(* IEC 61131-3 sources: com.logicals.lc3.webinar/RPMControl_Webinar/src_PRG_MQTT_Raspi2_ST, 4 files *)

(* ---- PRG_Raspi2_MQTTConnect.iecst ---- *)
/*
 * Raspi2
 * MQTTConnect Task
 */
PROGRAM PRG_Raspi2_MQTTConnect
   /*
    * PRG_Raspi2_MQTTConnect
    */
	VAR_EXTERNAL
    /*
     * Globaler TraceLevel
     */
     gui_TraceLevel : UINT;
	END_VAR
   /*
    * Status Verbindung zum Broker
    */
	VAR_EXTERNAL
		/*
		 * State und Channel vom Connect
		 */
		 MQTT_State   : MQTT_SUBSCRIBER_STATE;
		 MQTT_Channel : DINT;
	END_VAR

    VAR_EXTERNAL
        /*
         * Conecting Status an WebCon
         */
         gui_MQTTConnecting    : UINT; // Anzahl der Zyklen in MQTTConnecting
        /*
         * Conect und DisConnect Status an WebCon
         */
	     gui_MQTTConOkCycle    : UINT; // Anzahl der Zyklen bis MQTT Connect
	     gui_MQTTConNotOkCycle : UINT; // Anzahl der Zyklen wenn MQTT DisConnect
        /*
         * Conect Status an WebCon
         */
         gx_MQTTConOk      : BOOL;
    END_VAR

    VAR

    l_ConState : MQTT_SUBSCRIBER_STATE;

    l_RC       : MQTT_RC;
    ldi_Ch     : DINT;

    l_RC_Disconnect : MQTT_RC;

   END_VAR

   VAR
    /*
     * DiagnoseBits fuer RTS
     */
     lx_RTSInit     : BOOL;
     lx_RTSRun      : BOOL;
     lx_RTSShutDown : BOOL;
     lx_RTSTerm     : BOOL;
   END_VAR

   VAR
	 //
	 // Aus HCLib
     // Alle Verbindungen bedienen
     // Hier werden die Daten konkret verschickt!
     FB_Raspi2_MQTTConnect        : FB_MQTTConnect;
  END_VAR

  VAR
    /*
     * Der Datentyp enthaelt alle wesentlichen Informationen f�r die Basis-
     * Einstellungen von MQTT
     */
     l_MQTTInitKom    : DT_MQTT;
  END_VAR

 /*
  * Initialisierungsmerker
  */
  VAR
     FB_InitR_TRIG       : R_TRIG;
  END_VAR

  VAR
    /* Lokaler InitPuls im Baustein */
     lx_CycleInit : BOOL;

    /* Lokaler Puls im Baustein */
     lx_CyclePulse : BOOL;
    /* Lokaler Zyklustaktzaehler */
     li_CycleCount : INT;

    /* Lokaler InitZyklustaktzaehler */
     li_CycleCountInitVal : INT;
  END_VAR

  VAR
    lstr_PRGName      : STRING[30] := 'PRG_Raspi2_MQTTConnect';
    lui_TraceLevel    : UINT     := 5;

    lui_POU_UID       : UINT;                                      // Lokale POU-ID
    lstr_InstName     : STRING[30];
    lstr_POU_InstPath : STRING[128];                               // Lokale POU-ID
   END_VAR
 /*
  * -------------------------------------------------
  * Start SPS-Programm PRG_Raspi2_MQTTConnect
  * -------------------------------------------------
  */
 /*
  * InitZyklus setzen wenn MQTT aktiv gesetzt!
  */
  FB_InitR_TRIG(CLK := TRUE,Q => lx_CycleInit);

 /*
  * CyclePulse
  */
  lx_CyclePulse := NOT(lx_CyclePulse);

 /*
  * LifeTick bzw. ZyklusZaehler
  */
  li_CycleCount := li_CycleCount + 1;

   IF lx_CycleInit = TRUE THEN
       /*
        * Globalen TraceLevel uebernehmen
        */
       lui_TraceLevel := gui_TraceLevel;
      /*
       * PI-Name fuer GVL-Liste
       */
       lstr_InstName        := GET_CURRENT_PI_NAME();
       lstr_POU_InstPath    := lstr_PRGName;
       li_CycleCountInitVal := li_CycleCountInitVal + 1;
   END_IF;

    /*
     * Es wird ein MQTT_Connect aufgebaut
     * Wird fuer Publish/Subscribe verwendet!
     * NUR ein Connect je Resource zum Broker erlaubt!
     *
     * Im RTSTerm bzw. RTSShutdown MUSS der Connect Disconnected werden!
     */
     FB_Raspi2_MQTTConnect(vistr_InstPath                := lstr_InstName,
     	                    vistr_BrokerAddress          := l_MQTTInitKom.BrokerAdress,
                            vistr_ClientID               := l_MQTTInitKom.Raspi2ClientID,
                            vo_State                     => l_ConState,              // Status fuer Connect fuer alle zu oeffnenden Verbindungen (Pub/Sub) zum Broker
                            vo_RC                        => l_RC,                    // Status fuer Connect fuer alle zu oeffnenden Fehler (Pub/Sub) zum Broker
                            vodi_ch                      => ldi_Ch,                  // Status fuer Connect fuer alle zu oeffnenden Kanaele (Pub/Sub) zum Broker
                            voui_CycleCount_Connecting   => gui_MQTTConnecting,
                            voui_CycleCount_Connected    => gui_MQTTConOkCycle,      // Wert auch in WebCon
                            voui_CycleCount_NotConnected => gui_MQTTConNotOkCycle,   // Wert auch in WebCon
                            vox_MQTTConOk                => gx_MQTTConOk);           // Wert auch in WebCon
   /*
    * Ausgabe der Daten!
    */
    MQTT_State   := l_ConState;
    MQTT_Channel := ldi_ch;

   /*
    * Diagnosebits des RTS
    */
    RTSCycleInfo(Init     => lx_RTSInit,
  	             Run      => lx_RTSRun,
  	             Shutdown => lx_RTSShutDown,
  	             Term     => lx_RTSTerm);

   /*
    * Disconnect!
    * In RTS.CFG ShutDown Cycle von 3 Sekunden eintragen!
    */
    IF lx_RTSTerm = TRUE OR lx_RTSShutDown = TRUE THEN
     MQTT_Disconnect(ch := ldi_ch,
                     rc => l_RC_Disconnect);
     MQTT_State   := l_ConState;
     MQTT_Channel := -1;
    END_IF;

END_PROGRAM

(* ---- PRG_Raspi2_MQTTPublish_Header.iecst ---- *)
 /*
  * logi.cals GmbH
  * A-3100 St. Poelten
  * Europaplatz 7/1
  * Tel.: 0043-5-77147
  *
  * logi.cals automation solutions & services GmbH
  * D-40738 Langenfeld
  * Postfach 1306
  * Tel.: 0049-2173-91910
  *
  * Contact:
  * dieter.goltz@logicals.com
  *
  * History:
  * Created:
  * DG 2021-05-30 MQTT Header
  *
  * Modified:
  * DG 2021-05-30 MQTT Header
  */

 /*
  * Description
  * ===========
  */

 /*
  * Beschreibung
  * ============
  * MQTT Kommunikation
  * Publish Header
  *
  */

/*
 * Lokaler Test
 * ============
 * sudo mosquitto_sub -d -t test   - test = Name des Topic -> /Raspi2       - Header
 *                                                            /Raspi2/GV - Werte
 *
 * sudo mosquitto_pub -d -t test –m “Hello” - test = Name des Topic -> /Raspi2       - Header
 *                                                                     /Raspi2/?? - Werte
 *
 *                               -m "Hello" -> String der verschickt wird!
 */

/*
 * Publish des Header von Raspi2
 */
PROGRAM PRG_Raspi2_MQTTPublish_Header
    /*
	 * PRG_Raspi2_MQTTPublish_Header
	 */
    VAR_EXTERNAL
         MQTTHeader       : MQTTHeader;
    END_VAR

    VAR_EXTERNAL
      /*
       * Publish und Subsribe Status an WebCon
       */
	   gui_MQTTPublishOkCycle    : UINT; // Anzahl der Zyklen bis MQTT Publish
	   gui_MQTTSubscribeOkCycle  : UINT; // Anzahl der Zyklen wenn MQTT Subsribe

       gx_MQTTPublishState       : BOOL;

    END_VAR

	VAR_EXTERNAL
		/*
		 * State und Channel vom Connect
		 */
		 MQTT_State   : MQTT_SUBSCRIBER_STATE;
		 MQTT_Channel : DINT;
	END_VAR

	VAR_EXTERNAL
    /*
     * Globaler TraceLevel
     */
     gui_TraceLevel : UINT;
	END_VAR

	VAR_EXTERNAL
    /*
     * Uhrzeit und Daten von TimeBaustein abholen
     * und auf Globale Var in Byte schreiben
     * Fuer MQTT
     */
  	 gb_RTSSeconds : BYTE;
 	 gb_RTSMinutes : BYTE;
	 gb_RTSHours   : BYTE;

	 gb_RTSDay         : BYTE;
	 gb_RTSMonth       : BYTE;
	 gb_RTSYearHByte   : BYTE;
	 gb_RTSYearLByte   : BYTE;

    END_VAR

   VAR
      FB_MQTT_PublishRaspi2      : FB_MQTT_Publish;
   END_VAR

  VAR
    /*
     * Test Variablen um Publish zu untersuchen
     */
     lx_PublishHRaumOk    : BOOL := TRUE;
    /*
     * Test Publish
     */
     lx_TestMQTT     : BOOL := FALSE;
    /*
     * Publish Data (Header)
     * Wenn beide Optioenen FALSE sind, dann wird nicht geschickt
     * Wird im Code gesetzt!
     */
     lx_MQTTPublish  : BOOL := TRUE;

     lstr_PayLoad    : STRING[512];
     lMQTT_PayLoad   : STRING[512];
     l_TestPublishRC : MQTT_RC;
    /*
     * Der Datentyp enthaelt alle wesentlichen Initwerte f�r die MQTT-Kommunkation
     */
     l_MQTTInitKom         : DT_MQTT;
    /*
     * Status-Informationen
     */
     ldi_PublishLifeTick : DINT;
     lx_PublishOK        : BOOL;
     lui_IPVal1          : UINT;
     lui_IPVal2          : UINT;
     lui_IPVal3          : UINT;
     ldint_MQTTChannel   : DINT;
     ldint_MQTTCount     : DINT;
     ldint_MQTTrc        : DINT;
     lsint_MQTTState     : SINT;
     lx_MQTTENO          : BOOL;
     luint_MQTTLength    : UINT;
     lui_PubTick         : UINT;
  END_VAR

  VAR
    l_ConState : MQTT_SUBSCRIBER_STATE;
    ldi_ConCh  : DINT;
  END_VAR

  VAR
    lstr_PRGName   : STRING[30] := 'PRG_Raspi2_MQTTPublish_Header';
    lui_TraceLevel : UINT     := 5;
  END_VAR

  VAR
     FB_InitR_TRIG       : R_TRIG;
  END_VAR

  VAR
    /* Lokaler InitPuls im Baustein */
     lx_CycleInit : BOOL;

    /* Lokaler Puls im Baustein */
     lx_CyclePulse : BOOL;
    /* Lokaler Zyklustaktzaehler */
     li_CycleCount : INT;

    /* Lokaler InitZyklustaktzaehler */
     li_CycleCountInitVal : INT;
  END_VAR

 /*
  * InitZyklus setzen wenn MQTT aktiv gesetzt!
  */
  FB_InitR_TRIG(CLK := TRUE,Q => lx_CycleInit);
 /*
  * CyclePulse
  */
  lx_CyclePulse := NOT(lx_CyclePulse);

 /*
  * LifeTick bzw. ZyklusZaehler
  */
  li_CycleCount := li_CycleCount + 1;

  /*
   * Steuerung Publish / Subscribe ueber die Visu
   *
   * Publish
   * Welche Daten sollen an den Broker zurueckgeschickt werden
   * Subscribe
   * Welche Daten sollen geholt werden?
   */
   IF lx_CycleInit = TRUE THEN
      /*
       * Init Messages senden
       */
       lui_TraceLevel := gui_TraceLevel;
       li_CycleCountInitVal := li_CycleCountInitVal + 1;
   END_IF;
   /*
    * Daten von MQTTConnect
    */
    l_ConState := MQTT_State;
    ldi_ConCh  := MQTT_Channel;

    IF l_ConState = MQTT_SUBSCRIBER_STATE#CONNECTED THEN

   	   MQTTHeader.Second    := gb_RTSSeconds;
 	   MQTTHeader.Minute    := gb_RTSMinutes;
	   MQTTHeader.Hour      := gb_RTSHours;

	   MQTTHeader.Day       := gb_RTSDay;
	   MQTTHeader.Month     := gb_RTSMonth;
	   MQTTHeader.YearHByte := gb_RTSYearHByte;
	   MQTTHeader.YearLByte := gb_RTSYearLByte;

       MQTTHeader.IPVal3 := TO_BYTE(RIGHT(IN:= l_MQTTInitKom.Raspi2IPAdress, L := 1));
       MQTTHeader.IPVal2 := TO_BYTE(LEFT(RIGHT(IN:= l_MQTTInitKom.Raspi2IPAdress, L := 2),1));
       MQTTHeader.IPVal1 := TO_BYTE(LEFT(RIGHT(IN:= l_MQTTInitKom.Raspi2IPAdress, L := 3),1));

       FB_MQTT_PublishRaspi2(vi_MQTTHeader            := MQTTHeader,
                             vistr_IPAddr             := l_MQTTInitKom.Raspi2IPAdress,
                             vistr_BrokerIPAddr       := l_MQTTInitKom.BrokerAdress,
                             vix_Init                 := lx_CycleInit,
                             vi_State                 := l_ConState,
                             vdi_ch                   := ldi_ConCh,
       	                     vistr_BrokerPublishTopic := l_MQTTInitKom.Raspi2Topic,

                             vodi_PublishLifeTick    => ldi_PublishLifeTick,
                             vox_PublishOK           => lx_PublishOK,
                             voui_IPVal1             => lui_IPVal1,
                             voui_IPVal2             => lui_IPVal2,
                             voui_IPVal3             => lui_IPVal3,
                             vodint_MQTTChannel      => ldint_MQTTChannel,
                             vodint_MQTTCount        => ldint_MQTTCount,
                             vodint_MQTTrc           => ldint_MQTTrc,
                             vosint_MQTTState        => lsint_MQTTState,
                             vox_MQTTENO             => lx_MQTTENO,
                             vouint_MQTTLength       => luint_MQTTLength,
                             voui_PubTick            => lui_PubTick);

       gui_MQTTPublishOkCycle := TO_UINT(ldi_PublishLifeTick);
       gx_MQTTPublishState    := lx_PublishOK;

     END_IF;
END_PROGRAM

(* ---- PRG_Raspi2_MQTTPublish_IO.iecst ---- *)
 /*
  * logi.cals GmbH
  * A-3100 St. Poelten
  * Europaplatz 7/1
  * Tel.: 0043-5-77147
  *
  * logi.cals automation solutions & services GmbH
  * D-40738 Langenfeld
  * Postfach 1306
  * Tel.: 0049-2173-91910
  *
  * Contact:
  * dieter.goltz@logicals.com
  *
  * History:
  * Created:
  * DG 2021-05-30
  *
  * Modified:
  * DG 2021-05-30 IO
  */

 /*
  * Description
  * ===========
  */

 /*
  * Beschreibung
  * ============
  * MQTT Kommunikation
  * Publish Werte als Topics (IO)
  *
  * Austausch der aktuellen Daten mit dem Broker
  *
  */
 PROGRAM PRG_Raspi2_MQTTPublish_IO

   VAR_EXTERNAL
	    /* ProcessValue - Analogeingang_1 */
		gr_PV : REAL;
	    /* SetPoint     - Analogeingang_2 */
		gr_SP : REAL;
	    /* OutValue     - Analogausgang_1 */
		gr_Y : REAL;

	    /* ManualWert 0..100% */
		gr_Manual : REAL;

	    /* ProcessValue - Analogeingang_1 Skaliert 0..100%*/
		gr_PV_Scale : REAL;
	    /* SetPoint     - Analogeingang_2 Skaliert 0..100% */
		gr_SP_Scale : REAL;
	    /* OutValue     - Analogausgang_1 Skaliert 0..100% */
		gr_Ramp_In  : REAL;
        /*
         * Anzeige der Betriebsart 1Aus4
         */
        /* An Ausgang Ausgangswert = 0% */
        gx_ModeRPM0 : BOOL;
        /* An Ausgang Ausgangswert = 25% */
        gx_ModeRPM1 : BOOL;
        /* An Ausgang Ausgangswert = 50% */
        gx_ModeRPM2 : BOOL;
        /* An Ausgang SetPoint von Poti */
        gx_ModeRPM3 : BOOL;

       /*
        * Einstellwerte von Visu!
        * Per MQTT an TauriL / Raspi4
        */

       /*
        * Glaettung PT1-Verzoegerung
        */
        gr_PV_PT1_Set_T1 : REAL;

       /*
        * Regler Einstellungen
        * Per Regler-Task = 10ms Zyklszeit!
        */
        gr_PID_Set_TI  : REAL;
        gr_PID_Set_Kv  : REAL;
        gr_PID_Set_T1  : REAL;
        gr_PID_Set_Lvu : REAL;
        gr_PID_Set_Lvd : REAL;
        gr_PID_Set_Kp  : REAL;

       /*
        * Rampe Einstellungen fuer Regler
        */
        gr_Ramp_Set_OPC   : USINT;
        gr_Ramp_Set_SV    : REAL;
        gr_Ramp_Set_SpdUp : REAL;
        gr_Ramp_Set_SpdDn : REAL;
        gr_Ramp_Set_UpMax : REAL;
        gr_Ramp_Set_DnMax : REAL;
        gx_Ramp_Set_Stp   : BOOL;

        /* Blinkfunktion */
        gx_Flash : BOOL;
   END_VAR
  /*
   * PRG_Raspi2_MQTTPublish_IO
   */
   VAR_EXTERNAL
    /*
     * State und Channel vom Connect
     */
     MQTT_State   : MQTT_SUBSCRIBER_STATE;
     MQTT_Channel : DINT;
   END_VAR

   VAR_EXTERNAL
      /*
       * Globaler TraceLevel
       */
       gui_TraceLevel : UINT;
   END_VAR

  /*
   * Publish Topic / BOOL-Status von Topic
   */
   VAR
       FB_MQTT_Publish_IOBlink             : FB_MQTT_Publish_IO;

       FB_MQTT_Publish_IOModeRPM0       : FB_MQTT_Publish_IO;
       FB_MQTT_Publish_IOModeRPM1       : FB_MQTT_Publish_IO;
       FB_MQTT_Publish_IOModeRPM2       : FB_MQTT_Publish_IO;
       FB_MQTT_Publish_IOModeRPM3       : FB_MQTT_Publish_IO;

       FB_MQTT_Publish_IOValPID_TI      : FB_MQTT_Publish_IOVal;
       FB_MQTT_Publish_IOValPID_T1      : FB_MQTT_Publish_IOVal;
       FB_MQTT_Publish_IOValPID_KV      : FB_MQTT_Publish_IOVal;
       FB_MQTT_Publish_IOValPID_KP      : FB_MQTT_Publish_IOVal;

       FB_MQTT_Publish_IOValRMP_SpUp    : FB_MQTT_Publish_IOVal;
       FB_MQTT_Publish_IOValRMP_SpDn    : FB_MQTT_Publish_IOVal;
       FB_MQTT_Publish_IOValRMP_In      : FB_MQTT_Publish_IOVal;

   END_VAR

  VAR
    /*
     * Der Datentyp enthaelt alle wesentlichen Informationen fuer die Basis-
     * Einstellungen von MQTT
     */
     l_MQTTInitKom    : DT_MQTT;
  END_VAR

  VAR
    l_ConState : MQTT_SUBSCRIBER_STATE;
    ldi_ConCh  : DINT;
  END_VAR

   VAR
    lstr_PRGName : STRING[30] := 'PRG_Raspi2_MQTTPublish_IO';
    lui_TraceLevel : UINT     := 5;
   END_VAR
 /*
  * Initialisierungsmerker
  */
  VAR
     FB_InitR_TRIG       : R_TRIG;
  END_VAR

  VAR
    /* Lokaler InitPuls im Baustein */
     lx_CycleInit        : BOOL;

    /* Lokaler Puls im Baustein */
     lx_CyclePulse       : BOOL;
    /* Lokaler Zyklustaktzaehler */
     li_CycleCount       : INT;

    /* Lokaler InitZyklustaktzaehler */
     li_CycleCountInitVal : INT;
  END_VAR

  /*
   * InitZyklus setzen wenn MQTT aktiv gesetzt!
   */
   FB_InitR_TRIG(CLK := TRUE,Q => lx_CycleInit);

   lui_TraceLevel := gui_TraceLevel;

  /*
   * CyclePulse
   */
   lx_CyclePulse := NOT(lx_CyclePulse);

  /*
   * LifeTick bzw. ZyklusZaehler
   */
   li_CycleCount := li_CycleCount + 1;
  /*
   * -------------------------------------------------
   * Start SPS-Programm PRG_Raspi2_MQTTPublish_IO
   * -------------------------------------------------
   */

  /*
   * Steuerung Publish_IO
   *
   * Publish
   * Welche Einzel-Daten sollen an den Broker geschickt werden
   */
   IF lx_CycleInit = TRUE THEN
       li_CycleCountInitVal := li_CycleCountInitVal + 1;
   END_IF;

   /*
    * Daten von MQTTConnect
    */
    l_ConState := MQTT_State;
    ldi_ConCh  := MQTT_Channel;

   /*
    * Kommt von MQTTConnect
    * Wert MUSS 6 sein!
    */
    IF l_ConState = MQTT_SUBSCRIBER_STATE#CONNECTED /* connected */ THEN

   /*
    * Blinkfunktion
    */
    FB_MQTT_Publish_IOBlink(viui_TraceLevel            := lui_TraceLevel,
                            vix_PubIn                  := gx_Flash,
                            vistr_BrokerPublishTopicIO := l_MQTTInitKom.Raspi2TopicIOBlink,
                            vi_State                   := l_ConState,
                            vidi_Ch                    := ldi_ConCh);

   /*
    * Set Mode RPM 0 von Raspi2 per Publish
    */
    FB_MQTT_Publish_IOModeRPM0(viui_TraceLevel            := lui_TraceLevel,
                                  vix_PubIn                  := gx_ModeRPM0,
                                  vistr_BrokerPublishTopicIO := l_MQTTInitKom.Raspi2TopicIOModeRPM0,
                                  vi_State                   := l_ConState,
                                  vidi_Ch                    := ldi_ConCh);

   /*
    * Mode RPM 1 von Raspi2 per Publish
    */
    FB_MQTT_Publish_IOModeRPM1(viui_TraceLevel            := lui_TraceLevel,
                                  vix_PubIn                  := gx_ModeRPM1,
                                  vistr_BrokerPublishTopicIO := l_MQTTInitKom.Raspi2TopicIOModeRPM1,
                                  vi_State                   := l_ConState,
                                  vidi_Ch                    := ldi_ConCh);

   /*
    * Mode RPM 2 von Raspi2 per Publish
    */
    FB_MQTT_Publish_IOModeRPM2(viui_TraceLevel            := lui_TraceLevel,
                                  vix_PubIn                  := gx_ModeRPM2,
                                  vistr_BrokerPublishTopicIO := l_MQTTInitKom.Raspi2TopicIOModeRPM2,
                                  vi_State                   := l_ConState,
                                  vidi_Ch                    := ldi_ConCh);

   /*
    * Mode RPM 3 von Raspi2 per Publish
    */
    FB_MQTT_Publish_IOModeRPM3(viui_TraceLevel            := lui_TraceLevel,
                                  vix_PubIn                  := gx_ModeRPM3,
                                  vistr_BrokerPublishTopicIO := l_MQTTInitKom.Raspi2TopicIOModeRPM3,
                                  vi_State                   := l_ConState,
                                  vidi_Ch                    := ldi_ConCh);
   /*
    * PID-KP
    */
    FB_MQTT_Publish_IOValPID_KP(viui_TraceLevel            := lui_TraceLevel,
                            vir_PubIn                  := gr_PV,
                            vistr_BrokerPublishTopicIO := l_MQTTInitKom.Raspi2TopicIOPID_KP,
                            vi_State                   := l_ConState,
                            vidi_Ch                    := ldi_ConCh);

   /*
    * PID-KV
    */
    FB_MQTT_Publish_IOValPID_KV(viui_TraceLevel            := lui_TraceLevel,
                            vir_PubIn                  := gr_Y,
                            vistr_BrokerPublishTopicIO := l_MQTTInitKom.Raspi2TopicIOPID_KV,
                            vi_State                   := l_ConState,
                            vidi_Ch                    := ldi_ConCh);

   /*
    * PID-T1
    */
    FB_MQTT_Publish_IOValPID_T1(viui_TraceLevel            := lui_TraceLevel,
                                  vir_PubIn                  := gr_PID_Set_T1,
                                  vistr_BrokerPublishTopicIO := l_MQTTInitKom.Raspi2TopicIOPID_T1,
                                  vi_State                   := l_ConState,
                                  vidi_Ch                    := ldi_ConCh);

   /*
    * PID-TI
    */
    FB_MQTT_Publish_IOValPID_TI(viui_TraceLevel            := lui_TraceLevel,
                                  vir_PubIn                  := gr_PID_Set_TI,
                                  vistr_BrokerPublishTopicIO := l_MQTTInitKom.Raspi2TopicIOPID_TI,
                                  vi_State                   := l_ConState,
                                  vidi_Ch                    := ldi_ConCh);

   /*
    * Ramp Input = SetValue
    */
    FB_MQTT_Publish_IOValRMP_In(viui_TraceLevel            := lui_TraceLevel,
                                 vir_PubIn                  := gr_Ramp_In,
                                 vistr_BrokerPublishTopicIO := l_MQTTInitKom.Raspi2TopicIORMP_In,
                                 vi_State                   := l_ConState,
                                 vidi_Ch                    := ldi_ConCh);

   /*
    * Ramp_Speed Up
    */
    FB_MQTT_Publish_IOValRMP_SpUp(viui_TraceLevel            := lui_TraceLevel,
                                 vir_PubIn                  := gr_Ramp_Set_SpdUp,
                                 vistr_BrokerPublishTopicIO := l_MQTTInitKom.Raspi2TopicIORMP_SpUp,
                                 vi_State                   := l_ConState,
                                 vidi_Ch                    := ldi_ConCh);

   /*
    * Ramp Speed Dn
    */
    FB_MQTT_Publish_IOValRMP_SpDn(viui_TraceLevel            := lui_TraceLevel,
                                 vir_PubIn                  := gr_Ramp_Set_SpdDn,
                                 vistr_BrokerPublishTopicIO := l_MQTTInitKom.Raspi2TopicIORMP_SpDn,
                                 vi_State                   := l_ConState,
                                 vidi_Ch                    := ldi_ConCh);
   END_IF;

  END_PROGRAM

(* ---- PRG_Raspi2_MQTTSubscribe_Raspi4.iecst ---- *)
 /*
  * logi.cals GmbH
  * A-3100 St. Poelten
  * Europaplatz 7/1
  * Tel.: 0043-5-77147
  *
  * logi.cals automation solutions & services GmbH
  * D-40738 Langenfeld
  * Postfach 1306
  * Tel.: 0043-5-77147
  *
  * Contact:
  * dieter.goltz@logicals.com
  *
  * History:
  * Created:
  * DG 2021-05-05
  *
  * Modified:
  * DG 2021-02-09 Subscribe Daten Raspi4
  */

 /*
  * Description
  * ===========
  */

 /*
  * Beschreibung
  * ============
  * MQTT Kommunikation
  *
  * Subsribe der globalen Daten vom Broker
  *
  */

/*
 * MQTT Subscribe
 */
PROGRAM PRG_Raspi2_MQTTSubscribe_Raspi4

   VAR_EXTERNAL
     /*
      * Publish und Subsribe Status an WebCon
      */
	  gui_MQTTPublishOkCycle    : UINT; // Anzahl der Zyklen bis MQTT Publish
	  gui_MQTTSubscribeOkCycle  : UINT; // Anzahl der Zyklen wenn MQTT Subsribe

      gx_MQTTPublishState       : BOOL;

   END_VAR

   VAR_EXTERNAL
	    /* ProcessValue - Analogeingang_1 */
		gr_PV : REAL;
	    /* SetPoint     - Analogeingang_2 */
		gr_SP : REAL;
	    /* OutValue     - Analogausgang_1 */
		gr_Y : REAL;

	    /* ManualWert 0..100% */
		gr_Manual : REAL;

	    /* ProcessValue - Analogeingang_1 Skaliert 0..100%*/
		gr_PV_Scale : REAL;
	    /* SetPoint     - Analogeingang_2 Skaliert 0..100% */
		gr_SP_Scale : REAL;
	    /* OutValue     - Analogausgang_1 Skaliert 0..32767 */
		gr_Y_Scale  : REAL;
	    /* OutValue     - Regler Skaliert 0..100% */
		gr_PID_OUT  : REAL;
        /*
         * Anzeige der Betriebsart 1Aus4
         */
        /* An Ausgang Ausgangswert = 0% */
        gx_ModeRPM0 : BOOL;
        /* An Ausgang Ausgangswert = 25% */
        gx_ModeRPM1 : BOOL;
        /* An Ausgang Ausgangswert = 50% */
        gx_ModeRPM2 : BOOL;
        /* An Ausgang SetPoint von Poti */
        gx_ModeRPM3 : BOOL;

        /* Blinkfunktion */
        gx_Out8 : BOOL;
   END_VAR
    /*
	 * PRG_Raspi2_MQTTPublish
	 */
	VAR_EXTERNAL
    /*
     * Globaler TraceLevel
     */
     gui_TraceLevel : UINT;
	END_VAR
   /*
    * Status Verbindung zum Broker
    */
	VAR_EXTERNAL
		/*
		 * State und Channel vom Connect
		 */
		 MQTT_State   : MQTT_SUBSCRIBER_STATE;
		 MQTT_Channel : DINT;
	END_VAR

    VAR
	   /*
        * Der Datentyp enthaelt alle wesentlichen Initwerte fuer die MQTT-Kommunkation
        */
        l_MQTTInitKom  : DT_MQTT;
    END_VAR

    VAR
      /*
       * Raspi4
       */
       lx_Raspi4TopicOk1  : BOOL;
       lx_Raspi4TopicOk2  : BOOL;
       lx_Raspi4TopicOk3  : BOOL;
       lx_Raspi4TopicOk4  : BOOL;
       lx_Raspi4TopicOk5  : BOOL;
       lx_Raspi4TopicOk6  : BOOL;
       lx_Raspi4TopicOk7  : BOOL;
       lx_Raspi4TopicOk8  : BOOL;
       lx_Raspi4TopicOk9  : BOOL;
    END_VAR

    VAR
     lx_MQTTFlash : BOOL;

     lx_RPM1 : BOOL;
     lx_RPM2 : BOOL;
    END_VAR
	VAR
		ioImageRemote     : ARRAY [0..1023] OF BYTE;
		ioImageRemoteSize : DINT := 1024;
		ioImageRemoteLen  : DINT := -1;

	   /*
	    * Subscribe
	    */
		lx_CL1_subscribed  : BOOL := FALSE;  //

		rc_CL1  : MQTT_RC;

		lx_message_received : BOOL := FALSE;

		rc_ReceiveTopic     : MQTT_RC;

		lstr_ReceiveTopic   : STRING[255];

	   /*
	    * Alle erhaltenen Topics
	    * Array-Anpassung siehe TYPE END_TYPE Deklaration
	    */
		lstrarr_TopicArray : ARRAY [MQTT_MsgBound#Min..MQTT_MsgBound#Max] OF STRING[255];

	   /*
	    * Alle erhaltenen RC-Werte
	    */
		ldiarr_MessageRC   : ARRAY [MQTT_MsgBound#Min..MQTT_MsgBound#Max] OF DINT;
		larr_bImageRemote  : ARRAY [0..1023] OF BYTE;

	   /*
	    * Alle erhaltenen MessageLen-Werte
	    */
		ldiarr_MessageLen    : ARRAY [MQTT_MsgBound#Min..MQTT_MsgBound#Max] OF DINT;

       /*
        * Alle Messages
        */
		lstrarr_Messages     : ARRAY [MQTT_MsgBound#Min..MQTT_MsgBound#Max] OF STRING[1024];

		lusi_MessageIndex    : USINT := 0;
		lusi_MessageIndexMin : USINT := MQTT_MsgBound#Min;
		lusi_MessageIndexMax : USINT := MQTT_MsgBound#Max;
       /*
        * Raspi4
        */
		lui_Raspi4MessageLength1    : UINT;
		lui_Raspi4MessageLength2    : UINT;
		lui_Raspi4MessageLength3    : UINT;
		lui_Raspi4MessageLength4    : UINT;
		lui_Raspi4MessageLength5    : UINT;
		lui_Raspi4MessageLength6    : UINT;
		lui_Raspi4MessageLength7    : UINT;
		lui_Raspi4MessageLength8    : UINT;
		lui_Raspi4MessageLength9    : UINT;
       /*
        * Raspi4
        */
		lui_Raspi4MessageLifeTick1  : UINT;
		lui_Raspi4MessageLifeTick2  : UINT;
		lui_Raspi4MessageLifeTick3  : UINT;
		lui_Raspi4MessageLifeTick4  : UINT;
		lui_Raspi4MessageLifeTick5  : UINT;
		lui_Raspi4MessageLifeTick6  : UINT;
		lui_Raspi4MessageLifeTick7  : UINT;
		lui_Raspi4MessageLifeTick8  : UINT;
		lui_Raspi4MessageLifeTick9  : UINT;
       /*
        * Raspi4
        */
		ldi_Raspi4MessageRC1   : DINT;
		ldi_Raspi4MessageRC2   : DINT;
		ldi_Raspi4MessageRC3   : DINT;
		ldi_Raspi4MessageRC4   : DINT;
		ldi_Raspi4MessageRC5   : DINT;
		ldi_Raspi4MessageRC6   : DINT;
		ldi_Raspi4MessageRC7   : DINT;
		ldi_Raspi4MessageRC8   : DINT;
		ldi_Raspi4MessageRC9   : DINT;
       /*
        * Raspi4
        */
		lui_Raspi4MessagePosIdx1   : UINT;
		lui_Raspi4MessagePosIdx2   : UINT;
		lui_Raspi4MessagePosIdx3   : UINT;
		lui_Raspi4MessagePosIdx4   : UINT;
		lui_Raspi4MessagePosIdx5   : UINT;
		lui_Raspi4MessagePosIdx6   : UINT;
		lui_Raspi4MessagePosIdx7   : UINT;
		lui_Raspi4MessagePosIdx8   : UINT;
		lui_Raspi4MessagePosIdx9   : UINT;
	END_VAR

    VAR
      l_ConState : MQTT_SUBSCRIBER_STATE;
      ldi_Ch     : DINT;
    END_VAR

    VAR
      lstr_PRGName   : STRING[30] := 'PRG_Raspi2_MQTTSubscribe';
      lui_TraceLevel : UINT     := 5;
    END_VAR

   /*
    * Initialisierungsmerker
    */
    VAR
     FB_CycleInitR_TRIG       : R_TRIG;
    END_VAR

	VAR
	 li_CycleCount : INT;
	 lx_CyclePulse : BOOL;
	 lx_CycleInit  : BOOL;
	END_VAR

	FB_CycleInitR_TRIG(CLK := TRUE, Q => lx_CycleInit);
   /*
    * Laesst die Moeglichkeit zu den TraceLevel lokal zu aendern!
    */
    IF lx_CycleInit = TRUE THEN
	 lui_TraceLevel := gui_TraceLevel;
    END_IF;

    IF lx_CycleInit = TRUE THEN
	END_IF;

	li_CycleCount := li_CycleCount + 1;
	lx_CyclePulse := NOT lx_CyclePulse;

   /*
    * Interne Werte mit Uebergabe von MQTTConnect!
    */
	// MQTT_State := MQTT_GetState(ch := ldi_Ch, rc => rc, ENO => ENO);

    l_ConState := MQTT_State;
    ldi_ch     := MQTT_Channel;

	IF l_ConState = MQTT_SUBSCRIBER_STATE#CONNECTED THEN

		/* connect to topic in case connection has been established */
		IF NOT(lx_CL1_subscribed) THEN
           /*
            * Topics von Raspi4
            */
			MQTT_Subscribe(ch := ldi_Ch, topic := l_MQTTInitKom.Raspi4TopicIOBlink,       rc => rc_CL1); //
			MQTT_Subscribe(ch := ldi_Ch, topic := l_MQTTInitKom.Raspi4TopicIOPV_Scale,    rc => rc_CL1); //
			MQTT_Subscribe(ch := ldi_Ch, topic := l_MQTTInitKom.Raspi4TopicIOSP_Scale,    rc => rc_CL1); //
			MQTT_Subscribe(ch := ldi_Ch, topic := l_MQTTInitKom.Raspi4TopicIOY_Scale,     rc => rc_CL1); //
			MQTT_Subscribe(ch := ldi_Ch, topic := l_MQTTInitKom.Raspi4TopicIOPV,          rc => rc_CL1); //
			MQTT_Subscribe(ch := ldi_Ch, topic := l_MQTTInitKom.Raspi4TopicIOSP,          rc => rc_CL1); //
			MQTT_Subscribe(ch := ldi_Ch, topic := l_MQTTInitKom.Raspi4TopicIOY,           rc => rc_CL1); //
			MQTT_Subscribe(ch := ldi_Ch, topic := l_MQTTInitKom.Raspi4TopicIOModeRPM1,    rc => rc_CL1); //
			MQTT_Subscribe(ch := ldi_Ch, topic := l_MQTTInitKom.Raspi4TopicIOModeRPM2,    rc => rc_CL1); //

			lx_CL1_subscribed := rc_CL1 = MQTT_RC#OK;
		END_IF;

		// clear the receive ring buffer
		FOR lusi_MessageIndex := MQTT_MsgBound#Min TO MQTT_MsgBound#Max DO
		  lstrarr_Messages[lusi_MessageIndex] := '';
		END_FOR;

		/* if subscribed, obtain only the latest message */
		lx_message_received := FALSE;
		lusi_MessageIndex    := 0;

		REPEAT
			lstr_ReceiveTopic := MQTT_Receive(ch          := ldi_Ch,
                                              payload     := REF(ioImageRemote[0]),
                                              payload_len := ioImageRemoteSize,
                                              len         => ioImageRemoteLen,
                                              rc          => rc_ReceiveTopic);

			lx_message_received := TRUE;

			// convert the received byte array to a string
			lstrarr_Messages[lusi_MessageIndex] := StringFromByteArray(ioImageRemote, ioImageRemoteLen);
           /*
            * Das erhaltene Topic im Array hinterlegen
            */
            lstrarr_TopicArray[lusi_MessageIndex] := lstr_ReceiveTopic;
            ldiarr_MessageRC[lusi_MessageIndex]   := rc_ReceiveTopic;

			//
			// Messages-Index anpassen fuer weitere Nachrichten
			if (lusi_MessageIndex < lusi_MessageIndexMax) THEN
				lusi_MessageIndex := lusi_MessageIndex + 1;
			ELSE
				lusi_MessageIndex := lusi_MessageIndexMin;
			END_IF;

			IF rc_ReceiveTopic <> MQTT_RC#OK THEN
				EXIT;
			ELSE
			END_IF;

		UNTIL FALSE

		END_REPEAT;
	END_IF;

    lx_Raspi4TopicOk1  := FALSE;
    lx_Raspi4TopicOk2  := FALSE;
    lx_Raspi4TopicOk3  := FALSE;
    lx_Raspi4TopicOk4  := FALSE;
    lx_Raspi4TopicOk5  := FALSE;
    lx_Raspi4TopicOk6  := FALSE;
    lx_Raspi4TopicOk7  := FALSE;
    lx_Raspi4TopicOk8  := FALSE;
    lx_Raspi4TopicOk9  := FALSE;

   /*
    * Das Array der empfangenen Topics fuer Raspi4 analysieren
    */
    FOR lusi_MessageIndex := MQTT_MsgBound#Min TO MQTT_MsgBound#Max DO // 0 TO 20 DO
    /*
     * Raspi4
     */
     IF lstrarr_TopicArray[lusi_MessageIndex] = l_MQTTInitKom.Raspi4TopicIOBlink AND lx_Raspi4TopicOk1 = FALSE THEN
       lui_Raspi4MessagePosIdx1   := lusi_MessageIndex;
       lui_Raspi4MessageLifeTick1 := lui_Raspi4MessageLifeTick1 + 1;
       lui_Raspi4MessageLength1   := TO_UINT(ldiarr_MessageLen[lusi_MessageIndex]); // len(lstrarr_Messages[lusi_MessageIndex]);
       ldi_Raspi4MessageRC1       := ldiarr_MessageRC[lusi_MessageIndex];
       lx_Raspi4TopicOk1          := TRUE;

       IF lstrarr_Messages[lusi_MessageIndex] = 'TRUE' THEN
        lx_MQTTFlash := TRUE;
       ELSE
        lx_MQTTFlash := FALSE;
       END_IF;
     END_IF;
    /*
     * PV 0..100% (Anzeige BarGraph)
     */
     IF lstrarr_TopicArray[lusi_MessageIndex] = l_MQTTInitKom.Raspi4TopicIOPV_Scale  AND lx_Raspi4TopicOk2 = FALSE THEN
       lui_Raspi4MessagePosIdx2   := lusi_MessageIndex;
       lui_Raspi4MessageLifeTick2 := lui_Raspi4MessageLifeTick2 + 1;
       lui_Raspi4MessageLength2   := TO_UINT(ldiarr_MessageLen[lusi_MessageIndex]); // len(lstrarr_Messages[lusi_MessageIndex]);
       ldi_Raspi4MessageRC2       := ldiarr_MessageRC[lusi_MessageIndex];
       lx_Raspi4TopicOk2          := TRUE;
       gr_PV_Scale := TO_REAL(lstrarr_Messages[lusi_MessageIndex]);
     END_IF;
    /*
     * SetPoint 0..100% (Anzeige BarGraph)
     */
     IF lstrarr_TopicArray[lusi_MessageIndex] = l_MQTTInitKom.Raspi4TopicIOSP_Scale  AND lx_Raspi4TopicOk3 = FALSE THEN
       lui_Raspi4MessagePosIdx3   := lusi_MessageIndex;
       lui_Raspi4MessageLifeTick3 := lui_Raspi4MessageLifeTick3 + 1;
       lui_Raspi4MessageLength3   := TO_UINT(ldiarr_MessageLen[lusi_MessageIndex]); // len(lstrarr_Messages[lusi_MessageIndex]);
       ldi_Raspi4MessageRC3       := ldiarr_MessageRC[lusi_MessageIndex];
       lx_Raspi4TopicOk3          := TRUE;
       gr_SP_Scale := TO_REAL(lstrarr_Messages[lusi_MessageIndex]);
     END_IF;
    /*
     * Stellsignal 0..100% (Anzeige BarGraph)
     */
     IF lstrarr_TopicArray[lusi_MessageIndex] = l_MQTTInitKom.Raspi4TopicIOY AND lx_Raspi4TopicOk4 = FALSE THEN
       lui_Raspi4MessagePosIdx4   := lusi_MessageIndex;
       lui_Raspi4MessageLifeTick4 := lui_Raspi4MessageLifeTick4 + 1;
       lui_Raspi4MessageLength4   := TO_UINT(ldiarr_MessageLen[lusi_MessageIndex]); // len(lstrarr_Messages[lusi_MessageIndex]);
       ldi_Raspi4MessageRC4       := ldiarr_MessageRC[lusi_MessageIndex];
       lx_Raspi4TopicOk4          := TRUE;
       gr_PID_OUT := TO_REAL(lstrarr_Messages[lusi_MessageIndex]);
     END_IF;

    /*
     * RPM1
     */
     IF lstrarr_TopicArray[lusi_MessageIndex] = l_MQTTInitKom.Raspi4TopicIOModeRPM1 AND lx_Raspi4TopicOk5 = FALSE THEN
       lui_Raspi4MessagePosIdx5   := lusi_MessageIndex;
       lui_Raspi4MessageLifeTick5 := lui_Raspi4MessageLifeTick5 + 1;
       lui_Raspi4MessageLength5   := TO_UINT(ldiarr_MessageLen[lusi_MessageIndex]); // len(lstrarr_Messages[lusi_MessageIndex]);
       ldi_Raspi4MessageRC5       := ldiarr_MessageRC[lusi_MessageIndex];
       lx_Raspi4TopicOk5          := TRUE;

       IF lstrarr_Messages[lusi_MessageIndex] = 'TRUE' THEN
        lx_RPM1 := TRUE;
       ELSE
        lx_RPM1 := FALSE;
       END_IF;
        /* An Ausgang Ausgangswert = 50% */
        gx_ModeRPM1 := lx_RPM1;

     END_IF;

    /*
     * RPM2
     */
     IF lstrarr_TopicArray[lusi_MessageIndex] = l_MQTTInitKom.Raspi4TopicIOModeRPM1 AND lx_Raspi4TopicOk6 = FALSE THEN
       lui_Raspi4MessagePosIdx6   := lusi_MessageIndex;
       lui_Raspi4MessageLifeTick6 := lui_Raspi4MessageLifeTick6 + 1;
       lui_Raspi4MessageLength6   := TO_UINT(ldiarr_MessageLen[lusi_MessageIndex]); // len(lstrarr_Messages[lusi_MessageIndex]);
       ldi_Raspi4MessageRC6       := ldiarr_MessageRC[lusi_MessageIndex];
       lx_Raspi4TopicOk6          := TRUE;

       IF lstrarr_Messages[lusi_MessageIndex] = 'TRUE' THEN
        lx_RPM2 := TRUE;
       ELSE
        lx_RPM2 := FALSE;
       END_IF;
       /* An Ausgang Ausgangswert = 25% */
       gx_ModeRPM2 := lx_RPM2;
     END_IF;

    /*
     * Alle gefunden!
     */
     IF lx_Raspi4TopicOk1 = TRUE AND lx_Raspi4TopicOk2  = TRUE AND lx_Raspi4TopicOk3  = TRUE AND lx_Raspi4TopicOk4  = TRUE AND lx_Raspi4TopicOk5  = TRUE AND lx_Raspi4TopicOk6  = TRUE THEN
       lusi_MessageIndex := MQTT_MsgBound#Max;
     END_IF;

    END_FOR;

END_PROGRAM
